{attribute 'linkalways'} 
{attribute 'no_explicit_call' := 'This FB is a CLASS and must be accessed using methods or properties'}
{attribute 'enable_dynamic_creation'}
FUNCTION_BLOCK Node_ContainerType_Vector_TcVnVector3_INT EXTENDS Node
VAR
    out : _GUID;
END_VAR

METHOD PUBLIC  Clone : I_Node
VAR
	pNode : POINTER TO Node_ContainerType_Vector_TcVnVector3_INT;
END_VAR
pNode := __NEW(Node_ContainerType_Vector_TcVnVector3_INT);
Clone := pNode^;
END_METHOD

METHOD FB_init : BOOL
VAR_INPUT
	bInitRetains : BOOL; // if TRUE, the retain variables are initialized (warm start / cold start)
	bInCopyCode : BOOL;  // if TRUE, the instance afterwards gets moved into the copy code (online change)
END_VAR
AddOutput('out', out);
END_METHOD

METHOD PROTECTED OnExecute
out.Value := ContainerType_Vector_TcVnVector3_INT;
END_METHOD

END_FUNCTION_BLOCK

(* stored: Version 1.1.0.1, ProductVersion 3.1.4026.17
   POU Node_ContainerType_Vector_TcVnVector3_INT: Id {ef9829e7-ed6d-0cc3-15cd-7ec91e64445d}, SpecialFunc None
   Folder Constructor: Id {6cd192f0-1019-06fe-1ec3-234265e87ff9}
   Method Clone: Id {f25ec1e2-df80-0729-3b67-abc9b782c957}
   Method FB_init: Id {d6d2b9e0-8cb9-0f84-1b29-cc30dd74d7ae}
   Method OnExecute: Id {f3caae76-9d22-0543-3e98-7fe85ebd9206} *)
